Omron Sysmac Studio project TEST_HMI (Sysmac Studio 1.47.0.64008, StandardProject)

# Controller new_Controller_0: NX1P2-9024DT version 1.40
Task PrimaryTask (priority 4, period or condition 2000): Program0

VAR_GLOBAL
    start_00_hmi : BOOL;  (* published *)
    stop_00_hmi : BOOL;  (* published *)
    start_01_hmi : BOOL;  (* published *)
    stop_01_hmi : BOOL;  (* published *)
    start_02_hmi : BOOL;  (* published *)
    stop_02_hmi : BOOL;  (* published *)
    VAL_TIMER_0 : INT;  (* published *)
    VAL_TIMER_1 : INT;  (* published *)
    NX1P2_OUT_0 : BOOL;  (* at BuiltInIO://cpu/#0/Output_Bit_00; published *)
    NX1P2_OUT_1 : BOOL;  (* at BuiltInIO://cpu/#0/Output_Bit_01; published *)
    NX1P2_OUT_2 : BOOL;  (* at BuiltInIO://cpu/#0/Output_Bit_02; published *)
    NX1P2_OUT_3 : BOOL;  (* at BuiltInIO://cpu/#0/Output_Bit_03; published *)
    NX1P2_OUT_4 : BOOL;  (* at BuiltInIO://cpu/#0/Output_Bit_04; published *)
    NX1P2_OUT_5 : BOOL;  (* at BuiltInIO://cpu/#0/Output_Bit_05; published *)
    NX1P2_OUT_6 : BOOL;  (* at BuiltInIO://cpu/#0/Output_Bit_06; published *)
    NX1P2_OUT_7 : BOOL;  (* at BuiltInIO://cpu/#0/Output_Bit_07; published *)
    NX1P2_OUT_8 : BOOL;  (* at BuiltInIO://cpu/#0/Output_Bit_08; published *)
    NX1P2_OUT_9 : BOOL;  (* at BuiltInIO://cpu/#0/Output_Bit_09; published *)
END_VAR

PROGRAM Program0
VAR
    M0 : BOOL;
    LINT_00 : LINT;
    LINT_01 : LINT;
    TIMER_00 : TON;
    LINT_02 : LINT;
    VARIBLE_TIMER_00 : TIME;
    VARIBLE_TIMER_01 : TIME;
    TIMER_01 : TON;
    TIMER_03 : TON;
    TIMER_04 : TON;
    M1 : BOOL;
END_VAR
VAR_EXTERNAL
    start_00_hmi : BOOL;
    stop_00_hmi : BOOL;
    NX1P2_OUT_0 : BOOL;
    start_01_hmi : BOOL;
    stop_01_hmi : BOOL;
    NX1P2_OUT_1 : BOOL;
    NX1P2_OUT_2 : BOOL;
    VAL_TIMER_0 : INT;
    VAL_TIMER_1 : INT;
    NX1P2_OUT_3 : BOOL;
    NX1P2_OUT_4 : BOOL;
    start_02_hmi : BOOL;
    stop_02_hmi : BOOL;
END_VAR
VAR
    _p1 : BOOL;
    _p2 : BOOL;
END_VAR

(* Section Section0: ladder, written here as Structured Text *)

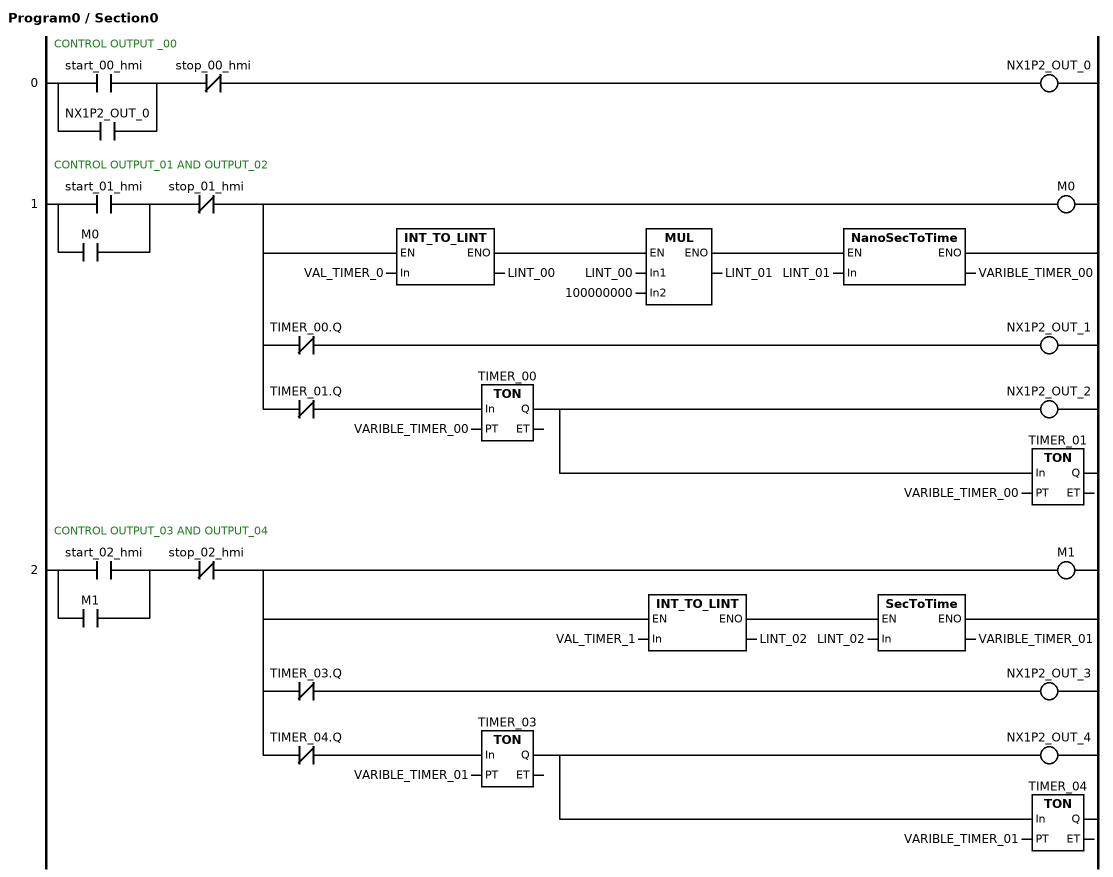
(* Rung 0: CONTROL OUTPUT _00 *)
NX1P2_OUT_0 := (start_00_hmi OR NX1P2_OUT_0) AND NOT stop_00_hmi;
(* Rung 1: CONTROL OUTPUT_01 AND OUTPUT_02 *)
_p1 := (start_01_hmi OR M0) AND NOT stop_01_hmi;
M0 := _p1;
IF _p1 THEN
    LINT_00 := INT_TO_LINT(In := VAL_TIMER_0);
    LINT_01 := LINT_00 * 100000000;
    VARIBLE_TIMER_00 := NanoSecToTime(In := LINT_01);
END_IF;
NX1P2_OUT_1 := _p1 AND NOT TIMER_00.Q;
TIMER_00(In := _p1 AND NOT TIMER_01.Q, PT := VARIBLE_TIMER_00);
NX1P2_OUT_2 := TIMER_00.Q;
TIMER_01(In := TIMER_00.Q, PT := VARIBLE_TIMER_00);
(* Rung 2: CONTROL OUTPUT_03 AND OUTPUT_04 *)
_p2 := (start_02_hmi OR M1) AND NOT stop_02_hmi;
M1 := _p2;
IF _p2 THEN
    LINT_02 := INT_TO_LINT(In := VAL_TIMER_1);
    VARIBLE_TIMER_01 := SecToTime(In := LINT_02);
END_IF;
NX1P2_OUT_3 := _p2 AND NOT TIMER_03.Q;
TIMER_03(In := _p2 AND NOT TIMER_04.Q, PT := VARIBLE_TIMER_01);
NX1P2_OUT_4 := TIMER_03.Q;
TIMER_04(In := TIMER_03.Q, PT := VARIBLE_TIMER_01);
END_PROGRAM